// TIA Portal V20 export
DATA_BLOCK "HMI变量汇总"   // DB10
{ S7_Optimized_Access := 'TRUE' }
// stored: MemoryReserve 100
   VAR
      Vis_Button_wideX1 : Bool;
      Vis_Button_wideX2 : Bool;
      Vis_Button_wideX3 : Bool;
      Vis_Button_wideX4 : Bool;
      Vis_Button_wideX5 : Bool;
      Vis_Button_wideX6 : Bool;
      Vis_Button_wideX7 : Bool;
      Vis_Button_wideX8 : Bool;
      Vis_Button_wideX9 : Bool;
      Vis_Button_wideX10 : Bool;
      Vis_Button_wideX11 : Bool;
      Vis_Button_wideX12 : Bool;
      Vis_Button_small1 : Bool;
      Vis_Button_small2 : Bool;
      Vis_Button_small3 : Bool;
      Vis_Button_small4 : Bool;
      Vis_Button_small5 : Bool;
      Vis_Button_small6 : Bool;
      Vis_Button_small7 : Bool;
      Vis_Button_small8 : Bool;
      Vis_Button_small9 : Bool;
      Vis_Button_small10 : Bool;
      Vis_Button_small11 : Bool;
      Vis_Button_small12 : Bool;
   END_VAR
BEGIN
END_DATA_BLOCK
